PROGRAM MAIN
VAR
{attribute 'pytmc' := '
        pv: PLC:113:TEST
'}
fbCoeRead : FB_Read70x1CoeData;

END_VAR

fbCoeRead(userNetId:='172.21.148.67.2.1');

END_PROGRAM

(* stored: Version 1.1.0.1, ProductVersion 3.1.4022.18
   POU MAIN: Id {37b0904a-2334-4b77-8e7e-d5a8d0d54da0}, SpecialFunc None *)
